{attribute 'linkalways'} 
{attribute 'no_explicit_call' := 'This FB is a CLASS and must be accessed using methods or properties'}
{attribute 'enable_dynamic_creation'}
FUNCTION_BLOCK _ETcWatchdogAccumulationType EXTENDS EnumDatatypeBase
VAR
	localData : ETcWatchdogAccumulationType;
	activeData : REFERENCE TO ETcWatchdogAccumulationType;
	enumBaseDatatype : _UINT(localData);
END_VAR

METHOD PRIVATE AddLocalEnumeration
VAR_INPUT
	Enumeration : T_MAXSTRING;
	Value : ETcWatchdogAccumulationType;
END_VAR
AddEnumeration(Enumeration, Value);
END_METHOD

PROPERTY PUBLIC Address : PVOID
GET
Address := ADR(activeData);
END_GET
END_PROPERTY

METHOD PUBLIC ClearReference
VAR_INPUT
END_VAR
activeData REF= localData;
SetBaseDatatypeReference();
END_METHOD

METHOD PUBLIC Clone : I_Datatype
VAR
    pClone : POINTER TO _ETcWatchdogAccumulationType;
END_VAR
pClone := __NEW(_ETcWatchdogAccumulationType(InitialValue := Value));
Clone := pClone^;
END_METHOD

METHOD FB_init : BOOL
VAR_INPUT
	bInitRetains : BOOL; // if TRUE, the retain variables are initialized (warm start / cold start)
	bInCopyCode : BOOL;  // if TRUE, the instance afterwards gets moved into the copy code (online change)
	InitialValue : ETcWatchdogAccumulationType;
END_VAR
localData := InitialValue;
AddBaseDatatype(enumBaseDatatype);
ClearReference();

AddLocalEnumeration('WD_ACC_TYPE_MEAN', ETcWatchdogAccumulationType.WD_ACC_TYPE_MEAN);
AddLocalEnumeration('WD_ACC_TYPE_PRODUCT', ETcWatchdogAccumulationType.WD_ACC_TYPE_PRODUCT);
END_METHOD

PROPERTY PUBLIC Identifier : T_MAXSTRING
GET
Identifier := 'ETcWatchdogAccumulationType';
END_GET
END_PROPERTY

METHOD IsEnumeratorValueEqual : BOOL
VAR_INPUT
	Enumerator : I_KeyValueForwardEnumerator;
END_VAR
VAR
	storedValue : ETcWatchdogAccumulationType;
END_VAR
IF NOT Enumerator.TryGet(storedValue) THEN
	RETURN;
END_IF

IsEnumeratorValueEqual := storedValue = activeData;
END_METHOD

METHOD PUBLIC MakeReferenceTo
VAR_INPUT
	ReferenceTarget : REFERENCE TO ETcWatchdogAccumulationType;
END_VAR
activeData REF= ReferenceTarget;
SetBaseDatatypeReference();
END_METHOD

METHOD PROTECTED SetBaseDatatypeReference
VAR_INPUT
END_VAR
enumBaseDatatype.MakeReferenceTo(activeData);
END_METHOD

PROPERTY PUBLIC Size : UDINT
GET
Size := SIZEOF(activeData);
END_GET
END_PROPERTY

METHOD TryMakeReferenceTo : BOOL
VAR_INPUT
	Target : I_Datatype;
END_VAR
VAR
	targetAsEnum : I_EnumDatatype;
	pTargetData : POINTER TO ETcWatchdogAccumulationType;
END_VAR
IF NOT Target.TryResolveAsEnumDatatype(targetAsEnum) THEN
	RETURN;
END_IF

IF targetAsEnum.Identifier <> Identifier THEN
	RETURN;
END_IF

pTargetData := Target.Address;
activeData REF= pTargetData^;
SetBaseDatatypeReference();
TryMakeReferenceTo := TRUE;
END_METHOD

PROPERTY PUBLIC Value : ETcWatchdogAccumulationType
GET
Value := activeData;
END_GET
SET
activeData := Value;
END_SET
END_PROPERTY

END_FUNCTION_BLOCK

(* stored: Version 1.1.0.1, ProductVersion 3.1.4024.12
   POU _ETcWatchdogAccumulationType: Id {be8674db-466e-48a1-84c7-c118d483c6f6}, SpecialFunc None
   Folder Constructor: Id {06f22b3a-1c01-47f5-a6d7-b8516b946eab}
   Folder Private: Id {0793f326-4fc2-40c8-acf1-e0d1aadd2a7a}
   Folder Protected: Id {06df1e93-0db5-455f-a4a0-a9b461669192}
   Method AddLocalEnumeration: Id {260828f6-c20c-4965-85d2-a9f18e65f1a8}
   Property Address: Id {3e2b9ae2-0a41-4e12-9d96-f17ea5f4a799}
   Get Get: Id {6661acf9-1dda-44d3-98b5-a0248f351071}
   Method ClearReference: Id {09b5b51d-bef8-4709-a96d-eb015ee4ba9c}
   Method Clone: Id {4d888f37-ebc8-438d-a347-168b51725a13}
   Method FB_init: Id {4246f205-0be5-487a-8f53-9a886de8ac98}
   Property Identifier: Id {2ef64ba6-95a1-4ec3-bb1d-0a184148e4ce}
   Get Get: Id {073bfedb-c420-41f7-8e8f-3c774d0e8377}
   Method IsEnumeratorValueEqual: Id {d123c1d9-d4f5-410b-83eb-5ccbcb07a477}
   Method MakeReferenceTo: Id {4f0de899-09ca-44ec-83ab-5bb3b4f3a454}
   Method SetBaseDatatypeReference: Id {c7b64c02-44cc-4c5f-8cdc-3b7394a8e2be}
   Property Size: Id {38e930b9-fd6f-4978-abc3-dd1e9b9b55be}
   Get Get: Id {9d0a25f0-8085-4871-b8bc-d350561af09b}
   Method TryMakeReferenceTo: Id {33b9e968-b590-4b37-8f92-6e4dd785c5de}
   Property Value: Id {15ad00ac-dda9-4979-b9d5-76b3136d7681}
   Get Get: Id {88fc820e-abea-4b0e-8749-3781f60bdf1f}
   Set Set: Id {ad39b36b-976d-4bab-af06-b6fadf1b4697} *)
